TYPE ST_PNInput_PeakShaveBox :
STRUCT
	w_Control			:	WORD;
	ui_FeedInCurrentLimit	:	UINT;
	ui_SupplyCurrentLimit	:	UINT;
	ui_VTRatio				:	UINT;
	UI_CTRatio				:	UINT;
END_STRUCT
END_TYPE

(* stored: Version 1.1.0.1, ProductVersion 3.1.4024.12
   DUT ST_PNInput_PeakShaveBox: Id {2411ed8f-5865-4a5f-80fb-4638b0cdc28b} *)
